(* PLC project 117_1_V0.5.project, CODESYS CODESYS V3.5 SP17 Patch 3 *)
(* stored: creationDateTime 1970-01-01T00:00:00, modificationDateTime 2026-03-26T18:14:32.4070562 *)

{attribute 'strict'}
TYPE DQ_VARS : (outPowerLightColumn, outRedLightColumn, outGreenLightColumn, outBuzzerLightColumn, outExciter, outRemoveLimitSwitch, outBit6, outBit7, outBit8, outBit9, outBit10, outBit11, outBit12, outBit13, outBit14, outBit15);
END_TYPE
